// TIA Portal V20 export
FUNCTION_BLOCK "FB_Fuellstand"   // FB23, LAD
{ S7_Optimized_Access := 'FALSE' }
AUTHOR : F.EE
VERSION : 1.2
// stored: AutoNumber false, SetENOAutomatically false
   VAR_INPUT
      iScaledMin : Real;
      iScaledMax : Real;
      iUnscaledMin : Real;
      iUnscaledMax : Real;
      iOffset : Real;
      iUnscaledAktVal : Word;
      iStoerungUnterdr : Bool;
      iQuittieren : Bool;
      iImpuls : Bool;
   END_VAR
   VAR_OUTPUT
      tOutStoe : "UDT_FuellstandStoe";
   END_VAR
   VAR_IN_OUT
      ioVisuSteuern : "UDT_FuellstandSteuern";
      ioVisuStatus : "UDT_FuellstandStatus";
   END_VAR
   VAR
      sZeitDrahtbruch : Real;
      sAktPos : Real;
      sAktPosGlatt : Real;
      sDrahtbruch : Bool;
      sZeitEinsch : Real;
      sZeitAussch : Real;
      sEinschalt : Bool;
      sAusschalt : Bool;
      sStoerBit1 : Bool;
      SWertAlt : Real;
      sHmStoerBit1 : Bool;
      sImStoerBit1 : Bool;
   END_VAR
   VAR_TEMP
      tOffset : Real;
      tVKE1 : Bool;
      tVKE0 : Bool;
      tbuffer01 : Real;
      tbuffer02 : Real;
      tbuffer03 : Real;
      tbuffer04 : Real;
      tbuffer05 : Real;
      tbufferDI01 : DInt;
      tbufferI01 : Int;
      tbufferI02 : Int;
      tbufferI03 : Int;
      tSaveDI : DInt;
      tRetVal : Int;
      tDrahtbruch : Bool;
   END_VAR
   VAR_TEMP   // added for the SCL form of the ladder/FBD networks
      _w1 : Bool;
      _w2 : Bool;
   END_VAR
BEGIN

REGION Network 2
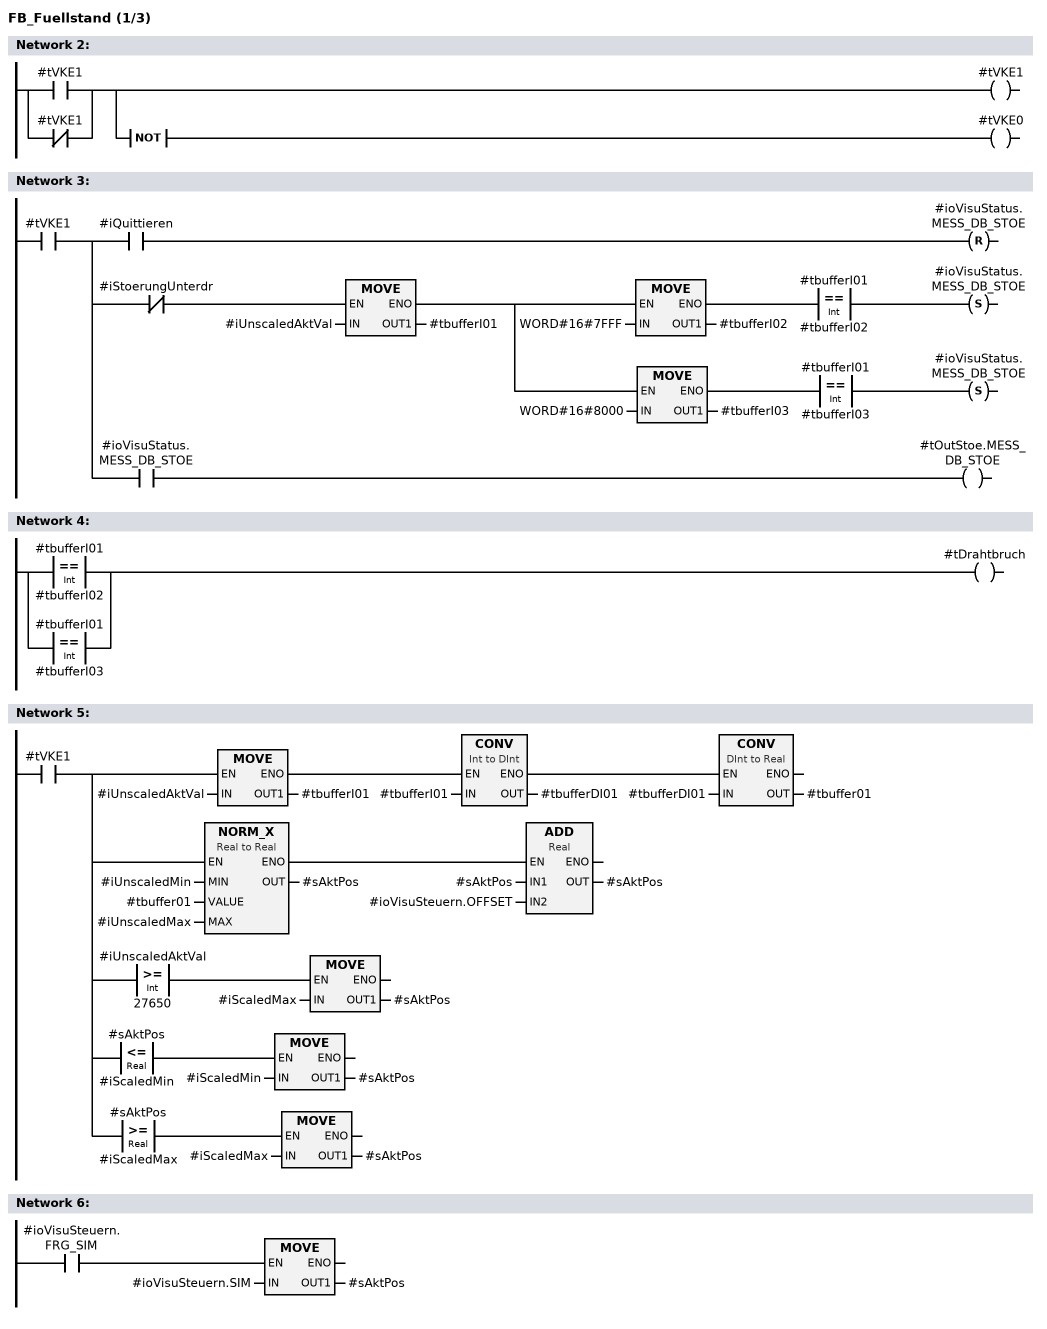
   RUNG wire#powerrail
      Contact( #tVKE1 )
      wire#w1
      Coil( #tVKE1 )
   END_RUNG
   RUNG wire#powerrail
      I_Contact( #tVKE1 )
   END_RUNG wire#w1
   RUNG wire#w1
      Not()
      Coil( #tVKE0 )
   END_RUNG
   // the same network as SCL:
   #tVKE1 := #tVKE1 OR NOT #tVKE1;
   #tVKE0 := NOT #tVKE1;
END_REGION

REGION Network 3
   RUNG wire#powerrail
      Contact( #tVKE1 )
      wire#w1
      Contact( #iQuittieren )
      R_Coil( #ioVisuStatus.MESS_DB_STOE )
   END_RUNG
   RUNG wire#w1
      I_Contact( #iStoerungUnterdr )
      { S7_GenerateENO := "TRUE" } Move(in := #iUnscaledAktVal, out1 => #tbufferI01)
      wire#w2
      { S7_GenerateENO := "TRUE" } Move(in := WORD#16#7FFF, out1 => #tbufferI02)
      { S7_Templates := "SrcType := Int" } EQ_Contact(in1 := #tbufferI01, in2 := #tbufferI02)
      S_Coil( #ioVisuStatus.MESS_DB_STOE )
   END_RUNG
   RUNG wire#w2
      { S7_GenerateENO := "TRUE" } Move(in := WORD#16#8000, out1 => #tbufferI03)
      { S7_Templates := "SrcType := Int" } EQ_Contact(in1 := #tbufferI01, in2 := #tbufferI03)
      S_Coil( #ioVisuStatus.MESS_DB_STOE )
   END_RUNG
   RUNG wire#w1
      Contact( #ioVisuStatus.MESS_DB_STOE )
      Coil( #tOutStoe.MESS_DB_STOE )
   END_RUNG
   // the same network as SCL:
   // ENO of a box is taken as its EN; it also drops when the box reports an error
   IF #tVKE1 AND #iQuittieren THEN #ioVisuStatus.MESS_DB_STOE := FALSE; END_IF;
   #_w1 := #tVKE1 AND NOT #iStoerungUnterdr;
   IF #_w1 THEN
       #tbufferI01 := #iUnscaledAktVal;
       #tbufferI02 := WORD#16#7FFF;
   END_IF;
   IF #_w1 AND (#tbufferI01 = #tbufferI02) THEN #ioVisuStatus.MESS_DB_STOE := TRUE; END_IF;
   IF #_w1 THEN #tbufferI03 := WORD#16#8000; END_IF;
   IF #_w1 AND (#tbufferI01 = #tbufferI03) THEN #ioVisuStatus.MESS_DB_STOE := TRUE; END_IF;
   #tOutStoe.MESS_DB_STOE := #tVKE1 AND #ioVisuStatus.MESS_DB_STOE;
END_REGION

REGION Network 4
   RUNG wire#powerrail
      { S7_Templates := "SrcType := Int" } EQ_Contact(in1 := #tbufferI01, in2 := #tbufferI02)
      wire#w1
      Coil( #tDrahtbruch )
   END_RUNG
   RUNG wire#powerrail
      { S7_Templates := "SrcType := Int" } EQ_Contact(in1 := #tbufferI01, in2 := #tbufferI03)
   END_RUNG wire#w1
   // the same network as SCL:
   #tDrahtbruch := (#tbufferI01 = #tbufferI02) OR (#tbufferI01 = #tbufferI03);
END_REGION

REGION Network 5
   RUNG wire#powerrail
      Contact( #tVKE1 )
      wire#w1
      { S7_GenerateENO := "TRUE" } Move(in := #iUnscaledAktVal, out1 => #tbufferI01)
      { S7_Templates := "[SrcType := Int, DestType := DInt]"; S7_GenerateENO := "TRUE" } Convert(in := #tbufferI01, out => #tbufferDI01)
      { S7_Templates := "[SrcType := DInt, DestType := Real]"; S7_GenerateENO := "TRUE" } Convert(in := #tbufferDI01, out => #tbuffer01)
   END_RUNG
   RUNG wire#w1
      { S7_Templates := "[SrcType := Real, DestType := Real]"; S7_GenerateENO := "TRUE" } Normalize(min := #iUnscaledMin, value := #tbuffer01, max := #iUnscaledMax, out => #sAktPos)
      { S7_Templates := "SrcType := Real"; S7_GenerateENO := "TRUE" } Add(in1 := #sAktPos, in2 := #ioVisuSteuern.OFFSET, out => #sAktPos)
   END_RUNG
   RUNG wire#w1
      { S7_Templates := "SrcType := Int" } GE_Contact(in1 := #iUnscaledAktVal, in2 := 27650)
      { S7_GenerateENO := "TRUE" } Move(in := #iScaledMax, out1 => #sAktPos)
   END_RUNG
   RUNG wire#w1
      { S7_Templates := "SrcType := Real" } LE_Contact(in1 := #sAktPos, in2 := #iScaledMin)
      { S7_GenerateENO := "TRUE" } Move(in := #iScaledMin, out1 => #sAktPos)
   END_RUNG
   RUNG wire#w1
      { S7_Templates := "SrcType := Real" } GE_Contact(in1 := #sAktPos, in2 := #iScaledMax)
      { S7_GenerateENO := "TRUE" } Move(in := #iScaledMax, out1 => #sAktPos)
   END_RUNG
   // the same network as SCL:
   // ENO of a box is taken as its EN; it also drops when the box reports an error
   IF #tVKE1 THEN
       #tbufferI01 := #iUnscaledAktVal;
       #tbufferDI01 := INT_TO_DINT(#tbufferI01);
       #tbuffer01 := DINT_TO_REAL(#tbufferDI01);
       #sAktPos := NORM_X(MIN := #iUnscaledMin, VALUE := #tbuffer01, MAX := #iUnscaledMax);
       #sAktPos := #sAktPos + #ioVisuSteuern.OFFSET;
   END_IF;
   IF #tVKE1 AND (#iUnscaledAktVal >= 27650) THEN #sAktPos := #iScaledMax; END_IF;
   IF #tVKE1 AND (#sAktPos <= #iScaledMin) THEN #sAktPos := #iScaledMin; END_IF;
   IF #tVKE1 AND (#sAktPos >= #iScaledMax) THEN #sAktPos := #iScaledMax; END_IF;
END_REGION

REGION Network 6
   RUNG wire#powerrail
      Contact( #ioVisuSteuern.FRG_SIM )
      { S7_GenerateENO := "TRUE" } Move(in := #ioVisuSteuern.SIM, out1 => #sAktPos)
   END_RUNG
   // the same network as SCL:
   IF #ioVisuSteuern.FRG_SIM THEN #sAktPos := #ioVisuSteuern.SIM; END_IF;
END_REGION

REGION Network 7
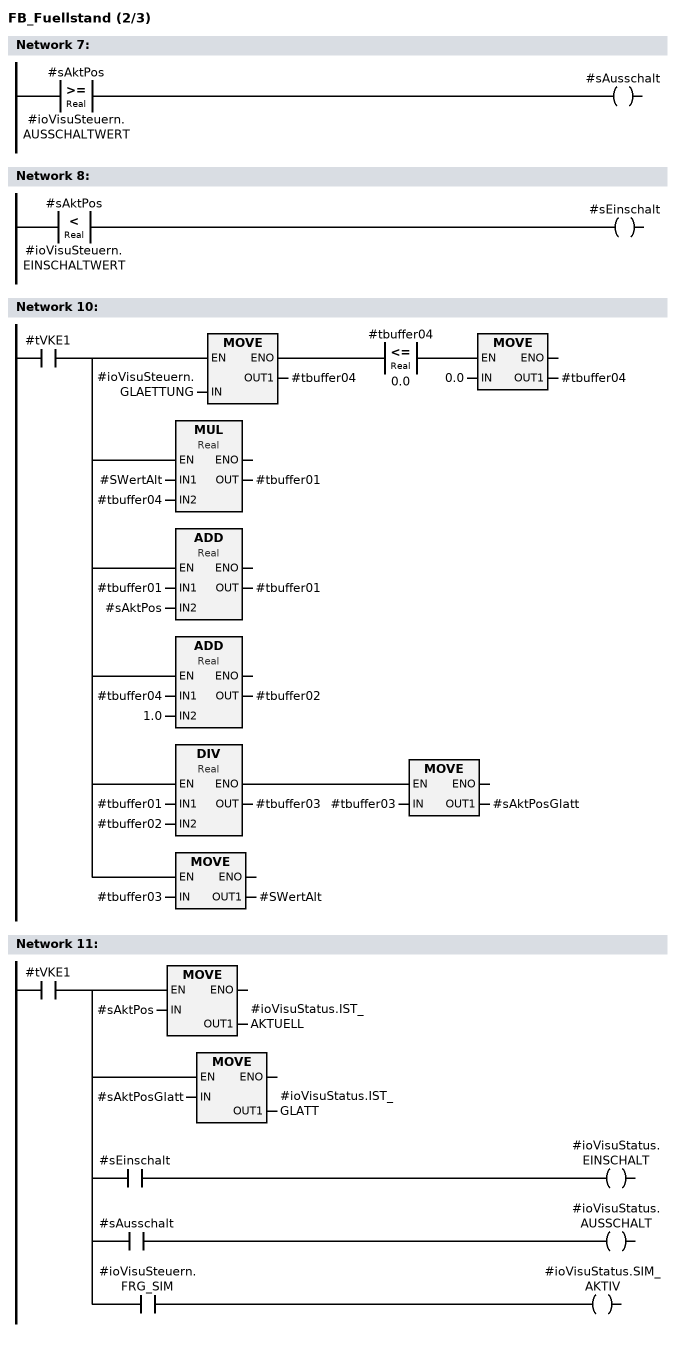
   RUNG wire#powerrail
      { S7_Templates := "SrcType := Real" } GE_Contact(in1 := #sAktPos, in2 := #ioVisuSteuern.AUSSCHALTWERT)
      Coil( #sAusschalt )
   END_RUNG
   // the same network as SCL:
   #sAusschalt := #sAktPos >= #ioVisuSteuern.AUSSCHALTWERT;
END_REGION

REGION Network 8
   RUNG wire#powerrail
      { S7_Templates := "SrcType := Real" } LT_Contact(in1 := #sAktPos, in2 := #ioVisuSteuern.EINSCHALTWERT)
      Coil( #sEinschalt )
   END_RUNG
   // the same network as SCL:
   #sEinschalt := #sAktPos < #ioVisuSteuern.EINSCHALTWERT;
END_REGION

REGION Network 9 (SCL)
   IF DINT_TO_DWORD(ROUND(#SWertAlt)) = 16#7FFFFFF THEN
       #SWertAlt := 0.0;
   END_IF;
END_REGION

REGION Network 10
   RUNG wire#powerrail
      Contact( #tVKE1 )
      wire#w1
      { S7_GenerateENO := "TRUE" } Move(in := #ioVisuSteuern.GLAETTUNG, out1 => #tbuffer04)
      { S7_Templates := "SrcType := Real" } LE_Contact(in1 := #tbuffer04, in2 := 0.0)
      { S7_GenerateENO := "TRUE" } Move(in := 0.0, out1 => #tbuffer04)
   END_RUNG
   RUNG wire#w1
      { S7_Templates := "SrcType := Real"; S7_GenerateENO := "TRUE" } Mul(in1 := #SWertAlt, in2 := #tbuffer04, out => #tbuffer01)
   END_RUNG
   RUNG wire#w1
      { S7_Templates := "SrcType := Real"; S7_GenerateENO := "TRUE" } Add(in1 := #tbuffer01, in2 := #sAktPos, out => #tbuffer01)
   END_RUNG
   RUNG wire#w1
      { S7_Templates := "SrcType := Real"; S7_GenerateENO := "TRUE" } Add(in1 := #tbuffer04, in2 := 1.0, out => #tbuffer02)
   END_RUNG
   RUNG wire#w1
      { S7_Templates := "SrcType := Real"; S7_GenerateENO := "TRUE" } Div(in1 := #tbuffer01, in2 := #tbuffer02, out => #tbuffer03)
      { S7_GenerateENO := "TRUE" } Move(in := #tbuffer03, out1 => #sAktPosGlatt)
   END_RUNG
   RUNG wire#w1
      { S7_GenerateENO := "TRUE" } Move(in := #tbuffer03, out1 => #SWertAlt)
   END_RUNG
   // the same network as SCL:
   // ENO of a box is taken as its EN; it also drops when the box reports an error
   IF #tVKE1 THEN #tbuffer04 := #ioVisuSteuern.GLAETTUNG; END_IF;
   IF #tVKE1 AND (#tbuffer04 <= 0.0) THEN #tbuffer04 := 0.0; END_IF;
   IF #tVKE1 THEN
       #tbuffer01 := #SWertAlt * #tbuffer04;
       #tbuffer01 := #tbuffer01 + #sAktPos;
       #tbuffer02 := #tbuffer04 + 1.0;
       #tbuffer03 := #tbuffer01 / #tbuffer02;
       #sAktPosGlatt := #tbuffer03;
       #SWertAlt := #tbuffer03;
   END_IF;
END_REGION

REGION Network 11
   RUNG wire#powerrail
      Contact( #tVKE1 )
      wire#w1
      { S7_GenerateENO := "TRUE" } Move(in := #sAktPos, out1 => #ioVisuStatus.IST_AKTUELL)
   END_RUNG
   RUNG wire#w1
      { S7_GenerateENO := "TRUE" } Move(in := #sAktPosGlatt, out1 => #ioVisuStatus.IST_GLATT)
   END_RUNG
   RUNG wire#w1
      Contact( #sEinschalt )
      Coil( #ioVisuStatus.EINSCHALT )
   END_RUNG
   RUNG wire#w1
      Contact( #sAusschalt )
      Coil( #ioVisuStatus.AUSSCHALT )
   END_RUNG
   RUNG wire#w1
      Contact( #ioVisuSteuern.FRG_SIM )
      Coil( #ioVisuStatus.SIM_AKTIV )
   END_RUNG
   // the same network as SCL:
   IF #tVKE1 THEN
       #ioVisuStatus.IST_AKTUELL := #sAktPos;
       #ioVisuStatus.IST_GLATT := #sAktPosGlatt;
   END_IF;
   #ioVisuStatus.EINSCHALT := #tVKE1 AND #sEinschalt;
   #ioVisuStatus.AUSSCHALT := #tVKE1 AND #sAusschalt;
   #ioVisuStatus.SIM_AKTIV := #tVKE1 AND #ioVisuSteuern.FRG_SIM;
END_REGION

REGION Network 12
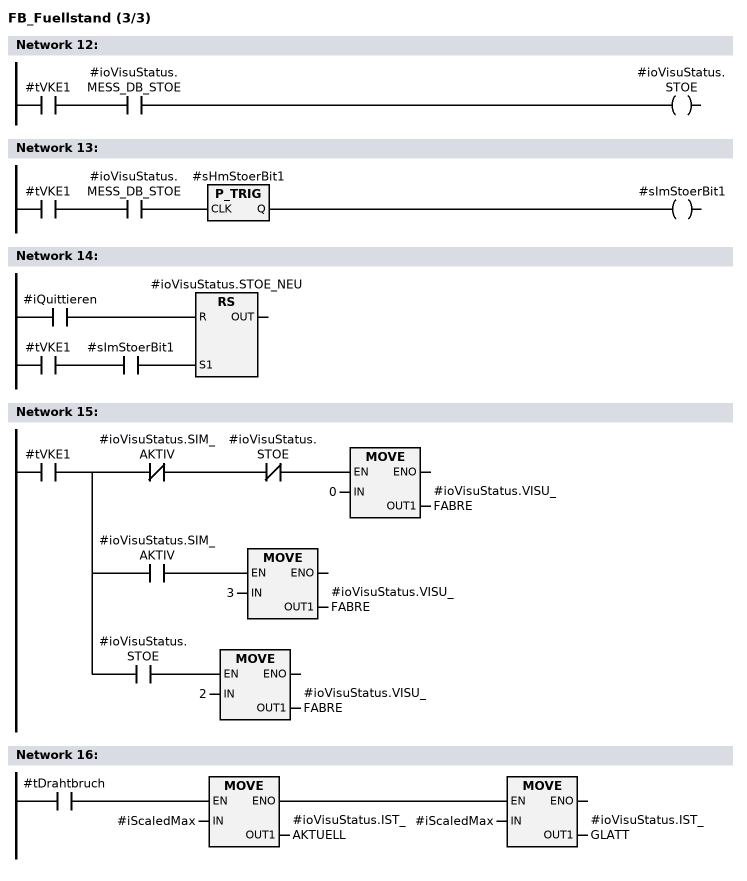
   RUNG wire#powerrail
      Contact( #tVKE1 )
      Contact( #ioVisuStatus.MESS_DB_STOE )
      Coil( #ioVisuStatus.STOE )
   END_RUNG
   // the same network as SCL:
   #ioVisuStatus.STOE := #tVKE1 AND #ioVisuStatus.MESS_DB_STOE;
END_REGION

REGION Network 13
   RUNG wire#powerrail
      Contact( #tVKE1 )
      Contact( #ioVisuStatus.MESS_DB_STOE )
      P_Trig( #sHmStoerBit1 )
      Coil( #sImStoerBit1 )
   END_RUNG
   // the same network as SCL:
   #_w1 := #tVKE1 AND #ioVisuStatus.MESS_DB_STOE;
   #_w2 := #_w1 AND NOT #sHmStoerBit1;   // rising edge
   #sHmStoerBit1 := #_w1;
   #sImStoerBit1 := #_w2;
END_REGION

REGION Network 14
   RUNG wire#powerrail
      Contact( #iQuittieren )
      S_RS(operand := #ioVisuStatus.STOE_NEU, s1 := wire#w1)
   END_RUNG
   RUNG wire#powerrail
      Contact( #tVKE1 )
      Contact( #sImStoerBit1 )
   END_RUNG wire#w1
   // the same network as SCL:
   IF #iQuittieren THEN
       #ioVisuStatus.STOE_NEU := FALSE;   // RS flip-flop
   END_IF;
   IF #tVKE1 AND #sImStoerBit1 THEN #ioVisuStatus.STOE_NEU := TRUE; END_IF;
END_REGION

REGION Network 15
   RUNG wire#powerrail
      Contact( #tVKE1 )
      wire#w1
      I_Contact( #ioVisuStatus.SIM_AKTIV )
      I_Contact( #ioVisuStatus.STOE )
      { S7_GenerateENO := "TRUE" } Move(in := 0, out1 => #ioVisuStatus.VISU_FABRE)
   END_RUNG
   RUNG wire#w1
      Contact( #ioVisuStatus.SIM_AKTIV )
      { S7_GenerateENO := "TRUE" } Move(in := 3, out1 => #ioVisuStatus.VISU_FABRE)
   END_RUNG
   RUNG wire#w1
      Contact( #ioVisuStatus.STOE )
      { S7_GenerateENO := "TRUE" } Move(in := 2, out1 => #ioVisuStatus.VISU_FABRE)
   END_RUNG
   // the same network as SCL:
   IF #tVKE1 AND NOT #ioVisuStatus.SIM_AKTIV AND NOT #ioVisuStatus.STOE THEN
       #ioVisuStatus.VISU_FABRE := 0;
   END_IF;
   IF #tVKE1 AND #ioVisuStatus.SIM_AKTIV THEN #ioVisuStatus.VISU_FABRE := 3; END_IF;
   IF #tVKE1 AND #ioVisuStatus.STOE THEN #ioVisuStatus.VISU_FABRE := 2; END_IF;
END_REGION

REGION Network 16
   RUNG wire#powerrail
      Contact( #tDrahtbruch )
      { S7_GenerateENO := "TRUE" } Move(in := #iScaledMax, out1 => #ioVisuStatus.IST_AKTUELL)
      { S7_GenerateENO := "TRUE" } Move(in := #iScaledMax, out1 => #ioVisuStatus.IST_GLATT)
   END_RUNG
   // the same network as SCL:
   // ENO of a box is taken as its EN; it also drops when the box reports an error
   IF #tDrahtbruch THEN
       #ioVisuStatus.IST_AKTUELL := #iScaledMax;
       #ioVisuStatus.IST_GLATT := #iScaledMax;
   END_IF;
END_REGION
END_FUNCTION_BLOCK
